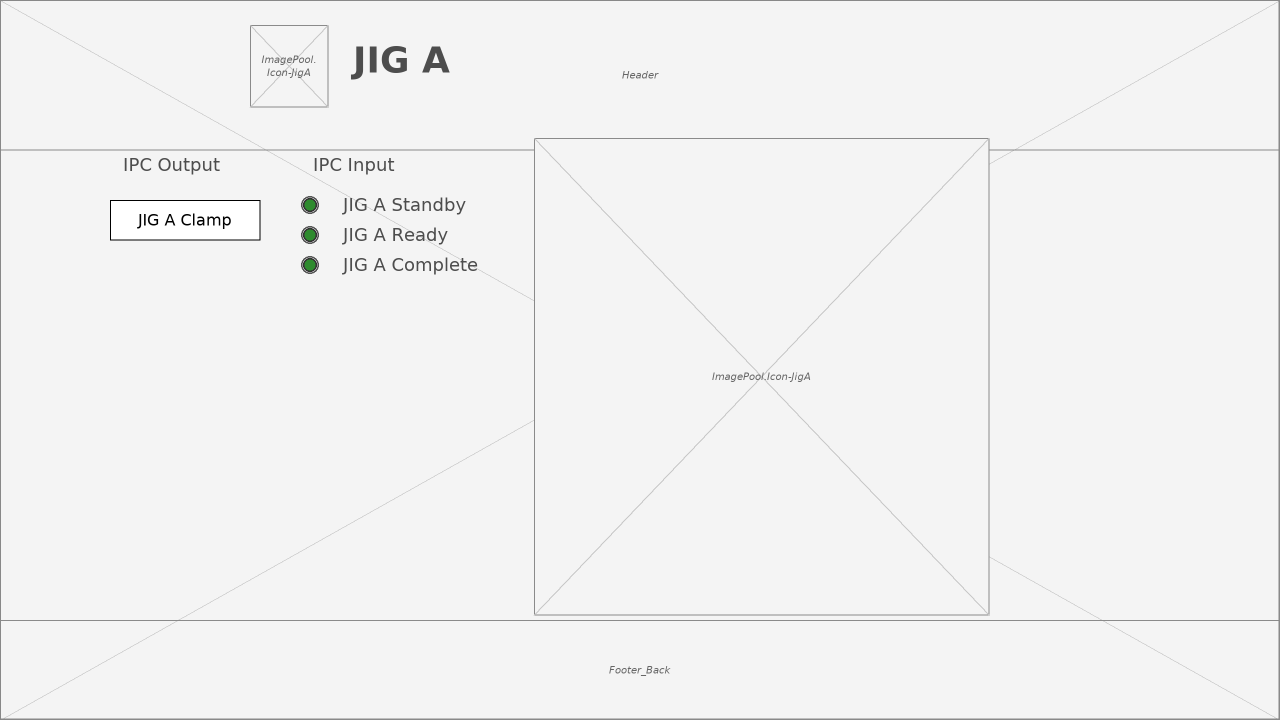
VISUALIZATION PAGE_JIG_A  // 1280x720
    Image (0,0 1280x720), image: ImagePool.The-New-Silver-Backgrounds
    Frame (0,620 1280x100)
        shows Footer_Back()
    Frame (0,0 1280x150)
        shows Header()
    Label (350,40 300x40), "JIG A"
    Label (120,150 150x30), "IPC Output"
    RoundedRectangle (110,200 150x40), "JIG A Clamp"
        toggle GVL.JIGA_Clamp
    Label (310,150 150x30), "IPC Input"
    Label (340,220 170x30), "JIG A Ready"
    Lamp1 (300,225 20x20), variable: GVL.JIGA_Ready, style: Lamp-Lamp1-Green
    Label (340,190 170x30), "JIG A Standby"
    Lamp1 (300,195 20x20), variable: GVL.JIGA_Standby, style: Lamp-Lamp1-Green
    Image (250,25 78x82), image: ImagePool.Icon-JigA
    Image (534,138 455x477), image: ImagePool.Icon-JigA
    Label (340,250 170x30), "JIG A Complete"
    Lamp1 (300,255 20x20), variable: GVL.JIGA_Complete, style: Lamp-Lamp1-Green
END_VISUALIZATION

(* stored: Version 1.1.0.1, ProductVersion 3.1.4024.12
   Visu PAGE_JIG_A: Id {f1cbe087-43a6-4da0-aa11-f2f1b01e03a2} *)
